ABB RAPID module: libMath.mod

MODULE libMath
    !*******************************************************************!
    ! Copyright (C) 2016 Piotr Ponikowski <pipon.github@gmail.com>      !
    !*******************************************************************!
    ! Module Name:  libMath                                             !
    ! Description:  math algorithms (basic & advanced)                  !
    ! Date:         2016-10-03                                          !
    ! Author:       Piotr Ponikowski <pipon.github@gmail.com>           !
    ! Contributors:                                                     !
    !*******************************************************************!

    !function used to calculate cross (scalar) product of two points (vectors)
    ! ret: pos = cross product result
    ! arg: vec1 - first point (vector)
    ! arg: vec2 - second point (vector)
    FUNC pos crossProd(pos vec1,pos vec2)
        RETURN [vec1.y*vec2.z-vec1.z*vec2.y,vec1.z*vec2.x-vec1.x*vec2.z,vec1.x*vec2.y-vec1.y*vec2.x];
    ENDFUNC

    !function used to set value of num depending of condition value
    ! ret: num = new value dependent of logical value
    ! arg: condition - logical value which determines output value
    ! arg: valTrue - output value if condition is true
    ! arg: valFalse - output value if condition is false
    FUNC num numLogicValue(bool condition,num valTrue,num valFalse)
        VAR num result:=0;

        IF condition THEN
            result:=valTrue;
        ELSE
            result:=valFalse;
        ENDIF

        RETURN result;
    ENDFUNC

    !function used to calc factorial
    ! ret: num = calculated factorial
    ! arg: val - input value
    FUNC num numFactorial(num val)
        VAR num result:=0;

        IF val=0 THEN
            result:=1;
        ELSE
            result:=val*numFactorial(val-1);
        ENDIF

        RETURN result;
    ENDFUNC

    !function used to check if selected value is inside set defined by upper and lower limit
    ! ret: bool = checked value is inside (TRUE) or outside (FALSE) of selected set
    ! arg: val - value to check
    ! arg: setStart - lower limit of checked set
    ! arg: setStop - upper limit of checked set
    FUNC bool numInsideSet(num val,num setStart,num setStop)
        RETURN val>=setStart AND val<=setStop;
    ENDFUNC

    !function used to check if selected value is outside set defined by upper and lower limit
    ! ret: bool = checked value is outside (TRUE) or inside (FALSE) of selected set
    ! arg: val - value to check
    ! arg: setStart - lower limit of checked set
    ! arg: setStop - upper limit of checked set
    FUNC bool numOutsideSet(num val,num setStart,num setStop)
        RETURN val<setStart OR val>setStop;
    ENDFUNC

    !function used to check selected parity type of inputted number
    ! ret: bool = inputted number is correct for user defined parity type
    ! arg: inputNum - number we want to check for parity
    ! arg: even - we want to check if number is even
    ! arg: odd - we want to check if number is odd
    FUNC bool numParity(num inputNum\switch even|switch odd)
        VAR bool result:=FALSE;

        !check what parity type we want to check
        IF Present(even) THEN
            !check if number is even
            result:=inputNum MOD 2=0;
        ELSEIF Present(odd) THEN
            !check if number is odd
            result:=inputNum MOD 2=1;
        ELSE
            !dont know what parity type to check
            result:=FALSE;
        ENDIF

        RETURN result;
    ENDFUNC

    !function used to generate random number
    ! ret: num = generated random number
    ! arg: setStart - lowest possible value (default: 0)
    ! arg: setEnd - highest possible value (default: 1)
    FUNC num numRandom(\num setStart\num setEnd\switch integer)
        VAR num result:=1;
        VAR num cStart:=0;
        VAR num cStop:=1;
        VAR num startValue;
        VAR num coeffA:=16807;
        VAR num coeffM:=8388608;

        !check user inputted data
        IF Present(setStart) cStart:=setStart;
        IF Present(setEnd) cStop:=setEnd;
        !check what kind of data user want
        IF Present(integer) THEN
            !integer - seed by time and use modulo
            result:=result*(GetTime(\Sec)/GetTime(\Min)+1);
            result:=Round(coeffA*result\Dec:=0) MOD coeffM;
            result:=cStart+(result MOD (cStop-cStart+1));
        ELSE
            !float - seed by time and cos to get values from 0 to 1
            result:=result*(GetTime(\Sec)+1);
            result:=result*(GetTime(\Min)+1);
            result:=cStart+(0.5+Cos(result)/2)*(cStop-cStart+1);
        ENDIF

        RETURN result;
    ENDFUNC

    !function used to get sign from inputted value
    ! ret: num = sign of value
    ! arg: val - value to check
    FUNC num numSign(num val)
        VAR num result:=0;

        IF val>0 result:=1;
        IF val<0 result:=-1;

        RETURN result;
    ENDFUNC

    !procedure used to swap two numbers
    ! arg: num1 - first number
    ! arg: num2 - second number
    PROC numSwap(INOUT num num1,INOUT num num2)
        VAR num temp;

        temp:=num1;
        num1:=num2;
        num2:=temp;
    ENDPROC

    !function used to calculate division of two orients
    ! ret: orient = division result
    ! arg: ori1 - first orient element (ORDER IMPORTANT!)
    ! arg: ori2 - second orient element (ORDER IMPORTANT!)
    FUNC orient oriDivide(orient ori1,orient ori2)
        RETURN NOrient(oriMult(ori1,oriInverse(ori2)));
    ENDFUNC

    !function used to calculate orient from pos (vector)
    ! ret: orient = calculated orient
    ! arg: point - pos (vector) to change
    FUNC orient oriFromPos(pos point)
        RETURN NOrient([0,point.x,point.y,point.z]);
    ENDFUNC

    !function used to calculate inversed orient
    ! ret: orient = inversed orient
    ! arg: ori - orient to inverse
    FUNC orient oriInverse(orient ori)
        !return negated orient components (Q1 not changed)
        RETURN NOrient([ori.q1,-ori.q2,-ori.q3,-ori.q4]);
    ENDFUNC

    !function used to multiply two orients
    ! ret: orient = result of multiplication
    ! arg: ori1 - first orient (ORDER IMPORTANT!)
    ! arg: ori2 - second orient (ORDER IMPORTANT!)
    FUNC orient oriMult(orient ori1,orient ori2)
        VAR orient result;

        result.q1:=ori1.q1*ori2.q1-ori1.q2*ori2.q2-ori1.q3*ori2.q3-ori1.q4*ori2.q4;
        result.q2:=ori1.q3*ori2.q4-ori1.q4*ori2.q3+ori1.q1*ori2.q2+ori1.q2*ori2.q1;
        result.q3:=ori1.q4*ori2.q2-ori1.q2*ori2.q4+ori1.q1*ori2.q3+ori1.q3*ori2.q1;
        result.q4:=ori1.q2*ori2.q3-ori1.q3*ori2.q2+ori1.q1*ori2.q4+ori1.q4*ori2.q1;

        RETURN result;
    ENDFUNC

    !function used to calulate distance from two positions
    ! ret: num = distance between poses
    ! arg: pose1 - first pose
    ! arg: pose2 - second pose
    FUNC num poseDistance(pose pose1,pose pose2)
        RETURN Distance(pose1.trans,pose2.trans);
    ENDFUNC

    !function used to calculate mid robt (and ortho shift it)
    ! ret: robtarget = middle robt (with ortho shift if needed)
    ! arg: robt1 - first robtarget
    ! arg: robt2 - second robtarget
    ! arg: orthoShift - otrhogonal shift length (if specified)
    FUNC robtarget robtCalcMidPnt(robtarget robt1,robtarget robt2\num orthoShift)
        VAR robtarget result;
        VAR pos vector;
        VAR pos orthoVector;
        VAR num dist:=0;

        !remeber orient,extax and config (pos will be changed below)
        result:=robt2;
        !calculate vector between robt1 and robt2
        vector:=vectorCalc(robt1.trans,robt2.trans);
        dist:=Distance(robt1.trans,robt2.trans);
        result:=shiftRobtByVector(result,vector,dist/2);
        !check if user want to otho sift this middle point
        IF Present(orthoShift) THEN
            orthoVector:=[-vector.y,vector.x,0];
            result:=shiftRobtByVector(result,orthoVector,orthoShift);
        ENDIF

        RETURN result;
    ENDFUNC

    !function used to calulate distance from two robtargets
    ! ret: num = distance between robtargets
    ! arg: robt1 - first robtarget
    ! arg: robt2 - second robtarget
    FUNC num robtDistance(robtarget robt1,robtarget robt2)
        RETURN Distance(robt1.trans,robt2.trans);
    ENDFUNC

    !function used to calculate the product of two robtargets
    ! ret: robtarget = product of two robtargets
    ! arg: robt1 - first robtarget to multiply (ORDER IMPORTANT!)
    ! arg: robt2 - second robtarget to multiply (ORDER IMPORTANT!)
    FUNC robtarget robtMult(robtarget robt1,robtarget robt2)
        VAR robtarget result;
        VAR pose tmpPose;

        !get external axes and robconf from first robtarget
        result:=robt1;
        !calculate multiply pose (abb function)
        tmpPose:=PoseMult(robtToPose(robt1),robtToPose(robt2));
        !cast pose result to robtarget
        result:=poseToRobt(tmpPose);

        RETURN result;
    ENDFUNC

    !procedure used to swap (change places) two robtargets
    ! arg: robt1 - first robtarget
    ! arg: robt2 - second robtarget
    PROC robtSwap(INOUT robtarget robt1,INOUT robtarget robt2)
        VAR robtarget tempRobt;

        tempRobt:=robt1;
        robT1:=robT2;
        robT2:=tempRobt;
    ENDPROC

    !function used to calculate angle between two vector
    ! ret: num = angle between vectors
    ! arg: vec - current vector
    ! arg: reference - reference vector
    FUNC num vectorAngle(pos vec,pos reference)
        VAR num result;
        VAR num numerator;
        VAR num denominator;

        !round two vectors to eliminate numerical errors
        vec:=roundPos(vec\posDec:=4);
        reference:=roundPos(reference\posDec:=4);
        !sprawdzamy czy te detale nie sa naprzeciw siebie
        IF vec.x=-reference.x AND vec.y=-reference.y THEN
            !detale sa naprzeciwko siebie = kat miedzy nimi 180
            result:=180;
        ELSEIF vec.x=reference.x AND vec.y=reference.y THEN
            !detale sa nalozone na siebie = kat miedzy nimi 0
            result:=0;
        ELSE
            !detale nie sa naprzeciwko - sprawdzamy kat miedzy nimi
            numerator:=DotProd(vec,reference);
            denominator:=VectMagn(vec)*VectMagn(reference);
            result:=ACos(numerator/denominator);
        ENDIF

        RETURN result;
    ENDFUNC

    !function used to check if selected vector is parallel to any axis
    ! ret: bool = inputted vector is parallel (TRUE) to any axis
    ! arg: vec - vector to check
    FUNC bool vectorAtAxis(pos vec)
        VAR bool result;
        VAR num ones:=0;

        !normalize vector to versor (length=1)
        vec:=vectorNorm(vec);
        !check if vector contains only one 1
        IF vec.x=1 Incr ones;
        IF vec.y=1 Incr ones;
        IF vec.z=1 Incr ones;
        !if there is only one 1 its OK (vector at axis)
        result:=ones=1;

        RETURN result;
    ENDFUNC

    !function used to caluclate vector definded by two pos
    ! ret: pos = znaleziony wektor
    ! arg: firstPos - pierwszy punkt (punkt poczatkowy wektora)
    ! arg: secondPos - drugi punkt (punkt koncowy wektora)
    FUNC pos vectorCalc(pos firstPos,pos secondPos\switch normalize)
        VAR pos result;

        !calculate vector
        result.x:=(secondPos.x-firstPos.x);
        result.y:=(secondPos.y-firstPos.y);
        result.z:=(secondPos.z-firstPos.z);
        !check if user wants to normalize
        IF Present(normalize) result:=vectorNorm(result);

        RETURN result;
    ENDFUNC

    !function used to count distance between vector and point
    ! ret: num = distance point <-> vector
    ! arg: vector - reference vector to count distance
    ! arg: point - point to count distance
    FUNC num vectorDistToPoint(pos vector,pos point)
        VAR num result:=-1;
        VAR pos tempVec{2};

        !wyznaczamy wektor od poczatku prostej do punktu
        tempVec{1}:=vectorCalc(point,vector);
        tempVec{2}:=vectorCalc(point,shiftPosByVector(vector,vector,100));
        !wyliczamy odleglosc
        result:=VectMagn(crossProd(tempVec{1},tempVec{2}))/VectMagn(vector);

        RETURN result;
    ENDFUNC

    !function used to inverse inputted vector
    ! ret: pos = vector inversed
    ! arg: vec - vector to inverse
    FUNC pos vectorInverse(pos vec)
        !return negated vector components
        RETURN [-vec.x,-vec.y,-vec.z];
    ENDFUNC

    !function used to normalize vector (versor)
    ! ret: pos = normalized vector (versor)
    ! arg: vec - vector to normalize
    FUNC pos vectorNorm(pos vec)
        VAR pos result;
        VAR num vecLen;

        !check vector length
        vecLen:=VectMagn(vec);
        !divide all components by vector length (to get versor)
        result.x:=vec.x/vecLen;
        result.y:=vec.y/vecLen;
        result.z:=vec.z/vecLen;

        RETURN result;
    ENDFUNC

    !function used to check if selected point is at the same side of vector as reference
    ! ret: bool = point is at the same side as reference (TRUE) or not (FALSE)
    ! arg: currPos - inputted point to check
    ! arg: ref - reference point
    ! arg: vecS - vector start point
    ! arg: vecE - vector end point
    FUNC bool vectorSameRefSide(pos currPos,pos ref,pos vecS,pos vecE)
        VAR bool result;
        VAR pos crossRes1;
        VAR pos crossRes2;

        crossRes1:=crossProd(vecE-vecS,currPos-vecS);
        crossRes2:=crossProd(vecE-vecS,ref-vecS);
        result:=DotProd(crossRes1,crossRes2)>=0;

        RETURN result;
    ENDFUNC
ENDMODULE
